// TIA Portal V16 export
// export: Created 2025-12-18T09:29:15.4872762Z, ExportSetting WithDefaults, DisplayName Totally Integrated Automation Portal, DisplayVersion V16, DisplayName TIA Portal Version Control Interface, DisplayVersion V16, DisplayName TIA Portal Openness, DisplayVersion V16, DisplayName STEP 7 Professional, DisplayVersion V16, DisplayName STEP 7 Safety, DisplayVersion V16, DisplayName WinCC Advanced, DisplayVersion V16
FUNCTION_BLOCK "StationConveyorControl"   // FB5, LAD
{ S7_Optimized_Access := 'TRUE' }
VERSION : 0.1
// stored: AutoNumber true, IsIECCheckEnabled false, IsRetainMemResEnabled false, MemoryReserve 100, SetENOAutomatically false, UDAEnableTagReadback false
   VAR_INPUT
      xEntrySensor { ExternalAccessible := 'False'; ExternalVisible := 'False'; ExternalWritable := 'False'} : Bool;
      xExitSensor { ExternalAccessible := 'False'; ExternalVisible := 'False'; ExternalWritable := 'False'} : Bool;
      xPositionerSensor { ExternalAccessible := 'False'; ExternalVisible := 'False'; ExternalWritable := 'False'} : Bool;
      xQueueSensor { ExternalAccessible := 'False'; ExternalVisible := 'False'; ExternalWritable := 'False'} : Bool;
      xInProcess : Bool;
   END_VAR
   VAR_IN_OUT
      xConveyor1 { ExternalAccessible := 'False'; ExternalVisible := 'False'; ExternalWritable := 'False'} : Bool;
      xConveyor2 { ExternalAccessible := 'False'; ExternalVisible := 'False'; ExternalWritable := 'False'} : Bool;
      xConveyor3 { ExternalAccessible := 'False'; ExternalVisible := 'False'; ExternalWritable := 'False'} : Bool;
   END_VAR
   VAR
      xMaterialAtExit : Bool;
      xMaterialAtPositioner : Bool;
      xProcessDone : Bool;
      xEdgeMemory1 { ExternalAccessible := 'False'; ExternalVisible := 'False'; ExternalWritable := 'False'} : Bool;
      xEdgeMemory2 { ExternalAccessible := 'False'; ExternalVisible := 'False'; ExternalWritable := 'False'} : Bool := false;
      xEdgeMemory3 { ExternalAccessible := 'False'; ExternalVisible := 'False'; ExternalWritable := 'False'} : Bool := false;
      xEdgeMemory4 { ExternalAccessible := 'False'; ExternalVisible := 'False'; ExternalWritable := 'False'} : Bool := false;
      xEdgeMemory5 : Bool;
   END_VAR
   VAR_TEMP   // added for the SCL form of the ladder/FBD networks
      _w1 : Bool;
      _w2 : Bool;
      _w3 : Bool;
   END_VAR
BEGIN

REGION Network 1
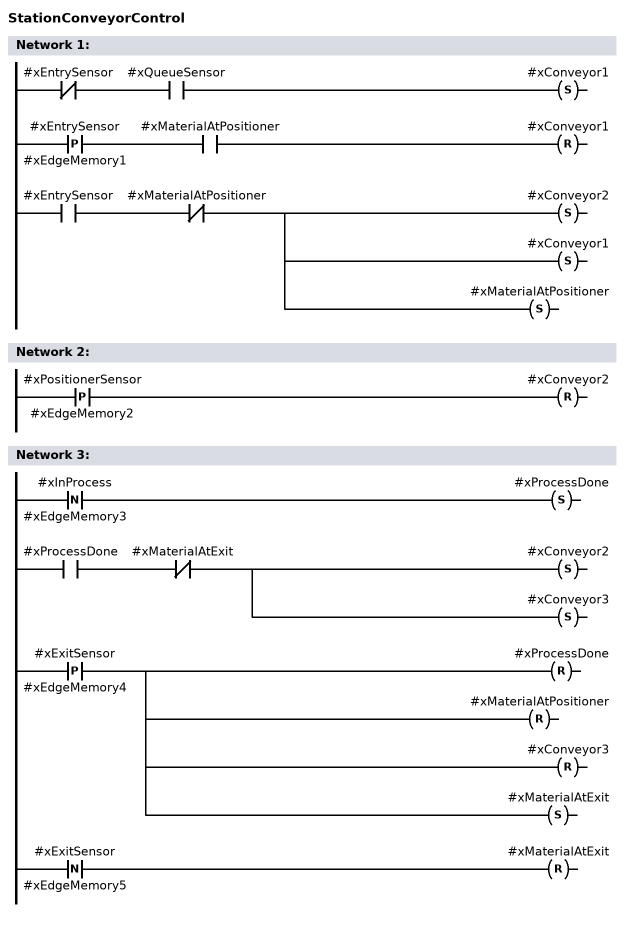
   RUNG wire#powerrail
      I_Contact( #xEntrySensor )
      Contact( #xQueueSensor )
      S_Coil( #xConveyor1 )
   END_RUNG
   RUNG wire#powerrail
      P_Contact(operand := #xEntrySensor, bit := #xEdgeMemory1)
      Contact( #xMaterialAtPositioner )
      R_Coil( #xConveyor1 )
   END_RUNG
   RUNG wire#powerrail
      Contact( #xEntrySensor )
      I_Contact( #xMaterialAtPositioner )
      wire#w1
      S_Coil( #xConveyor2 )
   END_RUNG
   RUNG wire#w1
      S_Coil( #xConveyor1 )
   END_RUNG
   RUNG wire#w1
      S_Coil( #xMaterialAtPositioner )
   END_RUNG
   // the same network as SCL:
   IF NOT #xEntrySensor AND #xQueueSensor THEN #xConveyor1 := TRUE; END_IF;
   #_w1 := #xEntrySensor AND NOT #xEdgeMemory1;   // rising edge of #xEntrySensor
   #xEdgeMemory1 := #xEntrySensor;
   IF #_w1 AND #xMaterialAtPositioner THEN #xConveyor1 := FALSE; END_IF;
   IF #xEntrySensor AND NOT #xMaterialAtPositioner THEN
       #xConveyor2 := TRUE;
       #xConveyor1 := TRUE;
       #xMaterialAtPositioner := TRUE;
   END_IF;
END_REGION

REGION Network 2
   RUNG wire#powerrail
      P_Contact(operand := #xPositionerSensor, bit := #xEdgeMemory2)
      R_Coil( #xConveyor2 )
   END_RUNG
   // the same network as SCL:
   #_w1 := #xPositionerSensor AND NOT #xEdgeMemory2;   // rising edge of #xPositionerSensor
   #xEdgeMemory2 := #xPositionerSensor;
   IF #_w1 THEN #xConveyor2 := FALSE; END_IF;
END_REGION

REGION Network 3
   RUNG wire#powerrail
      N_Contact(operand := #xInProcess, bit := #xEdgeMemory3)
      S_Coil( #xProcessDone )
   END_RUNG
   RUNG wire#powerrail
      Contact( #xProcessDone )
      I_Contact( #xMaterialAtExit )
      wire#w1
      S_Coil( #xConveyor2 )
   END_RUNG
   RUNG wire#w1
      S_Coil( #xConveyor3 )
   END_RUNG
   RUNG wire#powerrail
      P_Contact(operand := #xExitSensor, bit := #xEdgeMemory4)
      wire#w2
      R_Coil( #xProcessDone )
   END_RUNG
   RUNG wire#w2
      R_Coil( #xMaterialAtPositioner )
   END_RUNG
   RUNG wire#w2
      R_Coil( #xConveyor3 )
   END_RUNG
   RUNG wire#w2
      S_Coil( #xMaterialAtExit )
   END_RUNG
   RUNG wire#powerrail
      N_Contact(operand := #xExitSensor, bit := #xEdgeMemory5)
      R_Coil( #xMaterialAtExit )
   END_RUNG
   // the same network as SCL:
   #_w1 := NOT #xInProcess AND #xEdgeMemory3;   // falling edge of #xInProcess
   #xEdgeMemory3 := #xInProcess;
   IF #_w1 THEN #xProcessDone := TRUE; END_IF;
   IF #xProcessDone AND NOT #xMaterialAtExit THEN
       #xConveyor2 := TRUE;
       #xConveyor3 := TRUE;
   END_IF;
   #_w2 := #xExitSensor AND NOT #xEdgeMemory4;   // rising edge of #xExitSensor
   #xEdgeMemory4 := #xExitSensor;
   IF #_w2 THEN
       #xProcessDone := FALSE;
       #xMaterialAtPositioner := FALSE;
       #xConveyor3 := FALSE;
       #xMaterialAtExit := TRUE;
   END_IF;
   #_w3 := NOT #xExitSensor AND #xEdgeMemory5;   // falling edge of #xExitSensor
   #xEdgeMemory5 := #xExitSensor;
   IF #_w3 THEN #xMaterialAtExit := FALSE; END_IF;
END_REGION
END_FUNCTION_BLOCK
